TYPE Step :
(
	sleeping, 
	alarm, 
	snooze1, 
	snooze2, 
	wake, 
	toilet1,
	kitchen, 
	breakfast, 
	lunch, 
	toilet2, 
	garage, 
	cycling,
	train_check, 
	done	
) := sleeping;
END_TYPE

(* stored: Version 1.1.0.1, ProductVersion 3.1.4024.15
   DUT Step: Id {90e539c1-ea84-415e-b8f1-43acda1eeca4} *)
